Universal Robots PolyScope program: Pick_up_kettle.urp

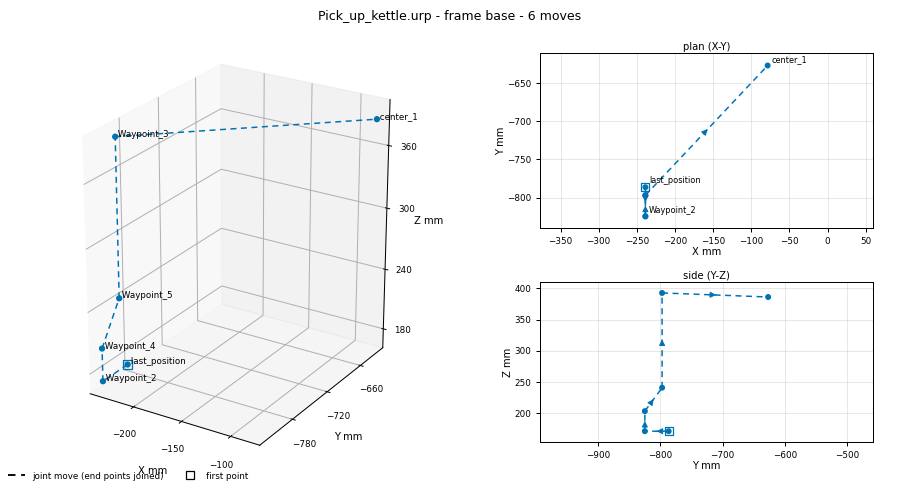
[picture p0: tool path of Pick_up_kettle.urp in frame base, 6 of 6 moves have a stored position in this frame; points joined in program order, loops and branches not executed]
Program Pick_up_kettle (installation=default directory=/programs/DMS createdIn=5.12.6.1102099 lastSavedIn=5.12.6.1102099 robotSerialNumber=20215500597)
Calibrated DH parameters: a=[0.000193, -0.066673, -0.391568, -0.000012, 0.00005, 0]; d=[0.162643, -472.05677, 465.132521, 7.058239, 0.099746, 0.099582]; alpha=[1.571116, 0.00089, 0.003862, 1.569269, -1.569248, 0]; deltaTheta=[0, -1.413394, 7.628392, 0.068187, 0, -0.000001]
Robot Program (runOnlyOnce=true)
  URCap Gripper (Robotiq_Grippers, Robotiq Inc.) dataModel(position=57.64705882352941, force=100.0, speed=64.0, positionInDouble=57.64705882352941, forceInDouble=100.0, speedInDouble=64.0, slaveIds=[9], blocking=true)
  MoveJ speed 60 deg/s, acceleration 80 deg/s^2 (useActiveTCP=true) feature=Base
    Waypoint last_position: TCP in base x=-238.783 y=-786.481 z=171.128 mm, rx=0.0287 ry=-2.2144 rz=2.2271 rad; joints [49.903, -56.994, 96.507, -40.117, 49.291, 179.673] deg; TCP offset x=0 y=0 z=191.5 mm, rx=0 ry=0 rz=0 rad
    Waypoint Waypoint_2: TCP in base x=-238.831 y=-824.668 z=171.125 mm, rx=0.0286 ry=-2.2144 rz=2.227 rad; joints [52.39, -53.216, 89.751, -37.121, 51.771, 179.65] deg
    URCap Gripper (Robotiq_Grippers, Robotiq Inc.) dataModel(position=80.25490196078431, force=100.0, speed=64.0, positionInDouble=80.25490196078431, forceInDouble=100.0, speedInDouble=64.0, slaveIds=[9], blocking=true)
    Waypoint Waypoint_4: TCP in base x=-238.8 y=-824.661 z=203.321 mm, rx=0.0286 ry=-2.2145 rz=2.227 rad; joints [52.392, -55.687, 88.397, -33.295, 51.76, 179.659] deg
    Waypoint Waypoint_5: TCP in base x=-238.804 y=-796.999 z=240.868 mm, rx=0.0286 ry=-2.2145 rz=2.227 rad; joints [50.62, -61.293, 91.299, -30.611, 49.981, 179.684] deg
    Waypoint Waypoint_3: TCP in base x=-238.809 y=-797.016 z=392.789 mm, rx=0.0285 ry=-2.2146 rz=2.2269 rad; joints [50.628, -68.308, 78.056, -10.362, 49.923, 179.708] deg
    Waypoint center_1: TCP in base x=-78.584 y=-626.961 z=386.266 mm, rx=0.0115 ry=-2.2034 rz=2.2303 rad; joints [53.978, -98.506, 113.326, -15.858, 53.984, 180.13] deg
